PROGRAM PRG_EpochConverter
//Convert Epoch to TimeStruct
VAR
	FileTime				: T_FILETIME;
	ConvertTime				: FB_SystemTimeToTzSpecificLocalTime;
END_VAR
VAR_INPUT
	IN_bIsWeird 			: BOOL; 				// Cas pour l'Epoch venant de Influx : offset de   82 011 087 
	IN_OffSet				: DINT :=  -82011087 ; 	// Cas pour l'Epoch venant de Influx : valeur de l'offset
	IN_Epoch				: LINT;					// Input 
END_VAR             		
VAR_OUTPUT          		
	OUT_TimeStruct_UTC		: TIMESTRUCT;
	OUT_TimeStruct_Local	: TIMESTRUCT;
END_VAR

IF IN_bIsWeird THEN
	IN_Epoch := IN_Epoch + IN_OffSet;
END_IF

FileTime.dwHighDateTime := LINT_TO_DWORD(SHR(IN_Epoch, 32));
FileTime.dwLowDateTime 	:= LINT_TO_DWORD(IN_Epoch);
OUT_TimeStruct_UTC 		:= FILETIME_TO_SYSTEMTIME( FileTime );
ConvertTime(in := OUT_TimeStruct_UTC, tzInfo := CstTimeZone_G, out => OUT_TimeStruct_Local);

END_PROGRAM

(* stored: Version 1.1.0.1, ProductVersion 3.1.4024.6
   POU PRG_EpochConverter: Id {7bdb086e-da8a-406c-b299-caee266fafa8}, SpecialFunc None *)
